Staubli VAL3: main.pgx

public program main()
  local tool l_tTool
  local num l_nSize
  local bool l_bSave
  local num l_nStatus
  local bool l_bToReset
  local bool l_bCalcolate
  local frame l_fNewWorld
begin
  // INIT
  call onStart()
  // LOOP UNTIL nKey=255
  do
    call tcp:getSize(l_nSize)
    call tcp:getTool(l_tTool,nIndexTool)
    call refresh()
    if l_bCalcolate
      $jogContext(l_tTool,world,0)
      l_bCalcolate=false
    endIf
    nKey=getKey()
    // tool setting

    // list....
    call use:listevent(nKey,nIndex,sEvent)
    nView=use:nView
    switch nKey
      case 263
        // BACKSPACE
        call onBackSpace(l_tTool)
        l_bCalcolate=true
        l_bSave=true
      break
      case 264
        // LEFT CLICK -1
        if nIndexTool>0
          nIndexTool=nIndexTool-1
          l_bSave=true
          l_bCalcolate=true
        endIf
      break
      case 268
        // RIGHT CLICK +1
        if nIndexTool<l_nSize-1
          nIndexTool=nIndexTool+1
          l_bSave=true
          l_bCalcolate=true
        endIf
      break
      case 271
        call onF1Event()
      break
      case 272
        call onF2Event()
      break
      case 273
        // HERE
        call onF3Event(l_bSave)
      break
      case 274
        // COMPUTE
        call onF4Event(l_bSave)
        l_bCalcolate=true
      break
      case 275
        // MOVE
        call onF5Event()
      break
      case 276
        // DUPLICATE
        call onF6Event(l_tTool.trsf,l_bSave)
      break
      case 277
        // DELETE
        call onF7Event(l_bSave)
      break
      case 278
        // NEW
        call onF8Event(l_bSave)
      break
      case 270
        // USE ALSO BACKSPACE
        // EDIT FIELD
        call onEnterEvent(l_tTool)
        l_bCalcolate=true
        l_bSave=true
      break
    endSwitch
    // release the resource
    delay(0)
  until nKey==255
  // on Exit
  $jogContext(l_tTool,world,0)
  call onExit(l_bSave)
end
